{attribute 'linkalways'} 
{attribute 'no_explicit_call' := 'This FB is a CLASS and must be accessed using methods or properties'}
{attribute 'enable_dynamic_creation'}
FUNCTION_BLOCK FINAL IntLiteralNode EXTENDS Node
VAR
	value : _INT(0);
	out : _INT(0);
END_VAR

METHOD PUBLIC Clone : I_Node
VAR
	pNode : POINTER TO IntLiteralNode;
END_VAR
pNode := __NEW(IntLiteralNode);
Clone := pNode^;
END_METHOD

METHOD FB_init : BOOL
VAR_INPUT
	bInitRetains : BOOL; // if TRUE, the retain variables are initialized (warm start / cold start)
	bInCopyCode : BOOL;  // if TRUE, the instance afterwards gets moved into the copy code (online change)
END_VAR
AddParameter('value', value);
AddOutput('out', out);
END_METHOD

METHOD PROTECTED OnExecute : HRESULT
VAR
END_VAR
out.value := value.value;
END_METHOD

END_FUNCTION_BLOCK

(* stored: Version 1.1.0.1, ProductVersion 3.1.4024.12
   POU IntLiteralNode: Id {fbb269dd-9577-0fa5-1c8c-18ea2c937326}, SpecialFunc None
   Folder Constructor: Id {5c7ca965-68e4-086b-3692-28cf7fd8d819}
   Method Clone: Id {a0452b7e-2208-021e-2b65-a65ea36a355c}
   Method FB_init: Id {444f5086-1aa2-0796-3a1e-ee02f28d629d}
   Method OnExecute: Id {9e05d5d1-0e0b-0dd7-048f-b54884cb0489} *)
